(* IEC 61131-3 sources: Everest-Indoor-Unit/SWNOVHIDUOUCR00/SWNOVHIDUOUCR00/Sources/Programs (part 2) *)

(* ---- 090_OutdoorUnitMng.st ---- *)
USING System;
USING System.Math;
USING Libs.Math;
USING Libs.Timer;

    VAR_GLOBAL
        (**Compressor speed when starting DHW*)
        DHW_InitRPS             : REAL;

    END_VAR

PROGRAM OutdoorUnitMng
    VAR
        (**Start/stop outdoor unit*)
        OU_OnOff                : BOOL;
        (**First DHW cycle*)
        DHW_FirstCycle          : BOOL;
        (**Outdoor unit cool/heat mode*)
        OU_CoolHeat             : BOOL;
    END_VAR

    IF RestoreDefault THEN
        RETURN;
    END_IF;

    OU_Unit.Info.Enabled := NOT(NoOutdoorUnit);
    OU_ComError := (NOT (OU_Unit.Info.isOnline)) AND NOT(NoOutdoorUnit);            //Communication error with outdoor unit

    IF(OU_Unit.Info.Enabled)THEN

        //Read OU values
        OU_OutsideTemp := OU_Unit.OutDoorTemp;
        OU_DscgP := OU_Unit.DscgP;
        OU_SuctP := OU_Unit.SuctP;
        OU_DscgTemp := OU_Unit.DscgTemp;
        OU_SuctTemp := OU_Unit.SuctTemp;
        OU_EnvZone := OU_Unit.EnvZone;
        OU_CompTemp := OU_Unit.CompTemp;
        OU_CurrSH := OU_Unit.CurrSH;
        OU_CurrDSH := OU_Unit.CurrDSH;
        OU_CurrSpd := OU_Unit.CurrSpd_RPS;
        OU_SHSetP := OU_Unit.CurrSHSetP;
        OU_CompOn := OU_Unit.CompOn;
        OU_CondTemp := OU_Unit.CondTemp;
        OU_EvapTemp :=  OU_Unit.EvapTemp;
        OU_CondInTemp := OU_Unit.CondInTemp;
        OU_CondOutTemp := OU_Unit.CondOutTemp;
        OU_WaterFlow := OU_Unit.WaterFlow;
        OU_HP_Status := OU_Unit.HP_Status;
        OU_CompMaxRps := Min(OU_Unit.MaxRPS, CompSpdMax);  //If there is a speed limitation to the compressor
        OU_RevValve := OU_Unit.RevValve;

        {REGION DHW SWITCH MANAGEMENT}

        //Store current information when going into DHW
        IF(OpState = OpStage_Status#DHW AND DHW_FirstCycle)THEN
            DHW_InitRPS      := OU_Unit.CurrSpd_RPS;
            FixedEBCount     := Ain_Data.Fct.ClimSupplyTemp;
            EBHP_Init        := EBHP;
            DHW_FirstCycle   := FALSE;
        ELSIF(NOT (OpState = OpStage_Status#DHW))THEN
            DHW_FirstCycle   := TRUE;
        END_IF;

        {ENDREGION}

        {REGION REQUEST MANAGER}
        //Manual mode
        IF(CompSpdMan > 0)THEN
            OU_OnOff := TRUE;
            OU_Req := MIN(CompSpdMan, OU_Unit.MaxRPS);
        ELSIF(UnitOff OR NoOutdoorUnit OR CompBlock)THEN //Unit off or outdoor unit not required
            OU_Req := 0;
            OU_OnOff := FALSE;
        ELSIF(OpState = OpStage_Status#DHW)THEN //DHW charge request
            IF(OU_Unit.CompOn AND DHW_InitRPS > 50.0)THEN //Keep compressor at steady speed if running at 50+ rps
                OU_OnOff := TRUE;

                IF(DHWBoost)THEN // Boost compressor speed during end of DHW
                    OU_Req := MIN(DHW_InitRPS + 30.0, OU_CompMaxRps);
                ELSE
                    OU_Req := DHW_InitRPS;
                END_IF;
            ELSE //DHW charge request locked at 50 rps
                OU_OnOff := TRUE;

                IF(DHWBoost)THEN // Boost compressor speed during end of DHW
                    OU_Req := MIN(50.0 + 30.0, OU_CompMaxRps);
                ELSE
                    OU_Req := MIN(50.0 , OU_CompMaxRps);
                END_IF;
            END_IF;
        ELSIF(OpState = OpStage_Status#HEATING AND SR_Energybalance_HP.Q1)THEN //Heating request
            OU_Req := ScalerLimited(PID_HeatReq, 0.0, 100.0, OU_Unit.MinRPS, OU_CompMaxRps);
            OU_OnOff := TRUE;

        ELSIF(OpState = Opstage_Status#COOLING AND SR_Energybalance_CH.Q1) THEN //Cooling request
            OU_Req := ScalerLimited(PID_CoolReq, 0.0, 100.0, OU_Unit.MinRPS, OU_CompMaxRps);
            OU_OnOff := TRUE;

        ELSE
            OU_Req := 0;
            OU_OnOff := TRUE;

        END_IF;
        {ENDREGION}

        //Write OU values
        OU_Unit.EEV_CompHeat    := OU_CompHeat;
        OU_Unit.CompReq         := OU_Req;
        OU_Unit.AlrmReset       := AlrmRes;
        OU_Unit.OnOff           := OU_OnOff;
        OU_Unit.Comp_MaxSpdLim  := CompSpdMax;
        OU_Unit.CoolHeat        := NOT CoolReq;// XOR SwToCoolReq;

        OU_Unit.SkipFreqBand1   := SkipFreqBand1 * 2;
        OU_Unit.SkipFreqBand2   := SkipFreqBand2 * 2;
        OU_Unit.SkipFreqBand3   := SkipFreqBand3 * 2;
        OU_Unit.SkipFreqF1      := SkipFreqF1 * 2;
        OU_Unit.SkipFreqF2      := SkipFreqF2 * 2;
        OU_Unit.SkipFreqF3      := SkipFreqF3 * 2;

        //Write new time
        OU_Unit.SetClock        := SetClock;
        OU_Unit.YearIn          := YearIn;
        OU_Unit.MonthIn         := MonthIn;
        OU_Unit.DayIn           := DayIn;
        OU_Unit.HourIn          := HourIn;
        OU_Unit.MinuteIn        := MinuteIn;
        OU_Unit.SecondsIn       := SecondIn;

    END_IF;

END_PROGRAM

(* ---- 100_PumpMng.st ---- *)
USING System;
USING System.Math;
USING Libs.Math;
USING Libs.PID_ADV;
USING Libs.Timer;
USING Libs.ExpFilt;

VAR_GLOBAL
    (**Actual PWM request heat medium pump*)
    Circ1Act_Req : REAL;
    DHWPumpReg : REAL;
END_VAR

PROGRAM PumpMng
    VAR

    END_VAR

    IF(PumpSpdGP1Man > 0)THEN    //Manual mode
        CircPmp_Req := TO_REAL(PumpSpdGP1Man);
    ELSIF(UnitOn) THEN    //Fixed pump speed for GP1 depending on current operating mode
//        IF OU_FreezeProtAct THEN
//            CircPmp_Req := PumpSpdFreezeProt;
        IF(OpState = OpStage_Status#DEFROST)THEN
            CircPmp_Req := PumpSpdDefrost;
        ELSIF(OpState = OpStage_Status#DHW)THEN
            CircPmp_Req := DHWChrgPumpSetPoint;
        ELSIF(OpState = OpStage_Status#HEATING) THEN
            CircPmp_Req := PumpspdHeatAuto;
        ELSIF(OpState = OpStage_Status#COOLING)THEN
            CircPmp_Req := PumpSpdCoolAuto;
        ELSE
            CircPmp_Req := 00.0;
        END_IF;
    ELSE
        CircPmp_Req := 0;
    END_IF;

    IF CircPmp_Req = 0 THEN // If pump shall be off the output shall be 97%
        Circ1Act_Req := 97;
    ELSE
    //Pump regulation
    Circ1Act_Req := Scaler(CircPmp_Req, 1, 100, 84, 10); //1-100 input is reversed and pump PWM input is scaled to fit the correct PWM curve.
    END_IF;

END_PROGRAM

(* ---- 110_HoursCounterMng.st ---- *)
USING System;
USING System.Math;
USING System.Timer;
USING Libs.Counters;

PROGRAM HoursCounterMng
    VAR
        (**Used for debug: n° of seconds for hour (Set 0=3600s)*)
        HrsCntrAdjust  : UINT;
        (**Source circuit 1 HoursCounter FB*)
        HrsCntr_Source1Circ1 : HoursCounter;
    END_VAR

    (*All the Programs are skipped while the default valeus are being installed*)
    IF RestoreDefault THEN
        RETURN;
    END_IF;

    (*--------------------------------
               HOURS COUNTER RESET
      --------------------------------*)
    IF ResTotCnt THEN
        ResTotCnt := FALSE;                                             (* Auto-Reset *)
    END_IF;
END_PROGRAM

(* ---- 950_GENERAL_MNG_END.st ---- *)
USING System.UI;

PROGRAM MainEnd
    {REGION WRITE BUFFER OF EACH SERIAL PORT}
    IF RetainRestored THEN
        //Stop all protocols.
        Supervisor.Stop();
        MBM_Line.Stop();
        Display.Stop();
    ELSE
        //Modbus Server line
        Supervisor.Write();
        //START COMMUNICATION
        Supervisor.Start();

        //Modbus Client line
        MBM_Line.Write();
        //START COMMUNICATION
        MBM_Line.Start();

        Display.Write();
    END_IF;

    {ENDREGION}

	(* Refresh UI *)
    SendVirtualKey(NO_KEY, 1);

END_PROGRAM

(* ---- 999_ExceptionManager.st ---- *)
USING System;
USING System.TEXT;

VAR_GLOBAL RETAIN INTERNAL
    (**Enable automatic test mode*)
    (*Allow to avoid the machine to stop in case of NFC/retain memory error.*)
    En_ATMode : BOOL;
END_VAR

PROGRAM ExceptionManager
    VAR_TEMP
        (**Event to read the error *)
        event           : Event;
        (**ID of task in error*)
        taskId          : INT;
        (**Error code*)
        error           : DINT;
        (**Erasures in case of retain/NFC written too often *)
        eraseures       : UDINT;
        (**Offset of erasure, in case of retain written too often *)
        eraseuresOffset : UDINT;
        (** Resume value: result of division by zero, square of negative, log of negative*)
        data            : UDINT := 0;
        (** Error string*)
        ErrorString     : STRING;
        (**Skip break of NFC/retain memory*)
        SkipRetainBreak : BOOL;
    END_VAR
    VAR_OUTPUT
        ExceptionError : DINT;
    END_VAR

    (*Get the event*)
    GetCurrentEvent(event);

    (*Check for a system error*)
    IF event.EventType = VMSystemEvent AND event.Mask = TO_DWORD(EVENT_EXCEPTION) THEN

        taskId := TO_INT(event.Data);
        GetLastTaskErrorCodeError(taskId, error);
        ExceptionError := error;

        ErrorString := FORMAT('Error 0x%08X ', error) + GetErrorDescription(error);

        (*Cause of error*)
        CASE error OF
            ERR_NFC_SAVE_TOO_OFTEN, ERR_RETAIN_SAVE_TOO_OFTEN :
                IF error = ERR_RETAIN_SAVE_TOO_OFTEN THEN
                    GetRetainInfo(eraseures, eraseuresOffset);
                ELSE
                    GetNfcInfo(eraseures, eraseuresOffset);
                END_IF;
                ErrorString := ErrorString + FORMAT(' Erasures for minute %d', eraseures);
                ErrorString := ErrorString + FORMAT(' Erasures offset %d', eraseuresOffset);

				SkipRetainBreak := En_ATMode;
        END_CASE;

        (*Write log*)
        WriteLog(LogLevel#Error_Level, ErrorString);

        (*Break in case of connection with STone*)
        IF IsDebuggerPresent() AND NOT(SkipRetainBreak) THEN
            SYSBREAK();
        END_IF;

        (*Resume the task, reset the task error*)
        ResumeTask(taskId, error, data);

        (** To reset after 30 seconds, enable the following define: *)
        {IF FALSE}
        HardwareReset(30, 0);
        {ENDIF}
	END_IF;

END_PROGRAM
